TYPE "TestSimple"
VERSION : 0.1
// Test UDT
   STRUCT
      TestBool : Bool;
      TestInt : Int;
      TestReal : Real;
   END_STRUCT;

END_TYPE
